// TIA Portal V16 export
// export: Created 2021-07-12T14:47:17.6616462Z, ExportSetting WithDefaults, DisplayName Totally Integrated Automation Portal, DisplayVersion V16, DisplayName TIA Portal Version Control Interface, DisplayVersion V16, DisplayName TIA Portal Openness, DisplayVersion V16, DisplayName STEP 7 Professional, DisplayVersion V16, DisplayName STEP 7 Safety, DisplayVersion V16, DisplayName WinCC Professional, DisplayVersion V16
VAR_GLOBAL   // PLC tag table "LSimaHydTO_Constants"
END_VAR
VAR_GLOBAL CONSTANT   // user constants
   LSIMAHYD_PROFILE_POINTS_UPPER_LIMIT : Int := 20;   // Upper limit of the points in the force profile
   LSIMAHYD_VCHAR_POINTS_UPPER_LIMIT : Int := 40;   // Upper limit of the points in the valve characteristic
END_VAR
